// TIA Portal project "TP1200" (V15)
// HMI za 12' zaslon

(* hardware
DEVICE "HMI_1"  TP1200 Comfort
   slot 0: "HMI_1"  TP1200 Comfort  6AV2 124-0MC01-0AX0  15.0.0.0
   slot 1: "HMI_RT_1"  TP1200 Comfort  6AV2 124-0MC01-0AX0  15.0.0.0
   slot 5: "HMI_1.IE_CP_1"  PROFINET Interface  15.0.0.0
      slot 1: "PROFINET Interface_1"  PROFINET Interface
         slot 1: "Port_1"  Port
         slot 2: "Port_2"  Port
   slot 7: "HMI_1.MPI/DP_CP_1"  MPI/DP Interface  15.0.0.0
*)

(* ===== HMI "HMI_RT_1" =====
system functions are stored by id; their names below are inferred from use

HMI tags "Default tag table"
   "Tag_ScreenNumber" : UInt, internal

graphic list "PAH": 0 'PAHmiruje_2'; 1 'PAHdeluje_2'

graphic list "MOTOR_SMER": 0 'MotorNaprej_1'; 1 'MotorNazaj_1'

graphic list "MOTOR_ON_OFF": 0 'MotorON_1'; 1 'MotorOFF'

graphic list "NACINI_DELOVANJA": 0..1 'Nastavitev_2'; 2..3 'ROC_1'; 4..5 'ROC_CIKEL_1'; 6..7 'AVT_NOZNO_2'; 8..9 'AVT_2'

screen "Root screen" 1280x800, template "Template_2"
   on GenerateScreen: SetTag("Tag_ScreenNumber", 1)

Template "Template_2" 1280x800
   GraphicView "Template_Graphic view_1" at 0,0 size 1277x800; Picture "root_template_3"
   IOField "Template_I/O field_1" at 1111,2 size 165x94; FormatPattern 999
   TextField "Template_Text field_1" at 529,48 size 224x52; Text 'RPM'
   TextField "Template_Text field_2" at 988,4 size 85x52; Text 'Text'
   GraphicView "Template_Graphic view_3" at 19,118 size 436x567; Picture "bruderer logo_2"
   Button "Template_Button_11" at 637,689 size 131x109; TextOff 'Text'
      on Click: function_efd93a16("ANAL.VHODI", 477, 157, -1, -1, 2)
   IOField "Template_I/O field_2" at 554,2 size 164x92; FormatPattern 999
   IOField "Template_I/O field_3" at 717,2 size 402x93; FormatPattern 999999
   Button "Template_Button_12" at 893,689 size 131x109; TextOff 'Text'
      on Click: function_efd93a16("DEBELINA", 477, 157, -1, -1, 2)
   Button "Template_Button_13" at 507,688 size 131x109; TextOff 'Text'
      on Click: function_efd93a16("DIG.VHODi", 477, 157, -1, -1, 2)
   Button "Template_Button_14" at 765,688 size 131x109; TextOff 'Text'
      on Click: function_efd93a16("DIG.IZHODI", 477, 157, -1, -1, 2)
   Button "Template_Button_15" at 380,689 size 131x109; TextOff 'Text'
      on Click: function_efd93a16("HOD", 477, 157, -1, -1, 2)
   Button "Template_Button_16" at 254,690 size 131x109; TextOff 'Text'
      on Click: function_efd93a16("PODAJALNA", 477, 157, -1, -1, 2)
   Button "Template_Button_17" at 129,690 size 131x109; TextOff 'Text'
      on Click: function_efd93a16("PAH", 477, 157, -1, -1, 2)
   Button "Template_Button_18" at 1022,688 size 131x109; TextOff 'Text'
      on Click: function_efd93a16("PODATKI", 477, 157, -1, -1, 2)
   Button "Template_Button_19" at 1145,687 size 131x109; TextOff 'Text'
      on Click: function_efd93a16("LISTANAPAK", 477, 157, -1, -1, 2)
   TextField "Template_Text field_3" at 719,5 size 401x44; Text 'ŠIFRA IZDELKA'
   TextField "Template_Text field_4" at 1121,58 size 151x44; Text 'RPM'
   Button "Template_Button_1" at 0,690 size 131x109; TextOff 'Text'
      on Click: function_efd93a16("stevci", 477, 157, -1, -1, 2)
   GraphicIOField "Template_Graphic I/O field_2" at 0,0 size 311x94; PictureList "NACINI_DELOVANJA"
   IOField "Template_I/O field_5" at 304,2 size 257x50; FormatPattern ????
   IOField "Template_I/O field_4" at 304,49 size 258x44; FormatPattern 99999999999999999999999999999999
   GraphicIOField "Graphic I/O field_2" at 1144,155 size 135x134; PictureList "MOTOR_SMER"
   GraphicIOField "Graphic I/O field_1" at 1144,290 size 135x134; PictureList "MOTOR_SMER"
   GraphicIOField "Graphic I/O field_3" at 1144,425 size 135x134; PictureList "PAH"

PopupScreen "PODATKI" 650x510
   GraphicView "Graphic view_1" at 0,0 size 649x510; Picture "ParametriOrodja"
   TextField "Text field_1" at 17,169 size 152x47; Text 'OZNAKA'
   TextField "Text field_2" at 16,240 size 153x41; Text 'POMIK'
   TextField "Text field_3" at 15,307 size 153x44; Text 'HOD'
   TextField "Text field_4" at 15,371 size 155x49; Text 'VIŠINA ORODJA'
   TextField "Text field_5" at 389,375 size 152x43; Text 'HIT. PODAJANJA'
   TextField "Text field_6" at 390,302 size 156x49; Text 'POSPEŠEK'
   TextField "Text field_9" at 388,237 size 159x45; Text 'PODLOGA ZGORAJ'
   TextField "Text field_10" at 389,169 size 154x44; Text 'PODLOGA SPODAJ'
   TextField "Text field_11" at 17,439 size 155x49; Text 'SPROSITEV'

PopupScreen "PODAJALNA" 650x510
   GraphicView "Graphic view_1" at 0,0 size 649x510; Picture "PodajalnikTraku_1"

PopupScreen "PAH" 650x510
   GraphicView "Graphic view_1" at 0,0 size 649x510; Picture "VisinaPaha"

PopupScreen "LISTANAPAK" 650x510
   GraphicView "Graphic view_1" at 0,0 size 649x510; Picture "ListaNapak_2"

PopupScreen "HOD" 650x510
   GraphicView "Graphic view_1" at 0,0 size 649x510; Picture "HOD"

PopupScreen "DIG.VHODi" 650x510
   GraphicView "Graphic view_1" at 0,0 size 649x510; Picture "DI_1"

PopupScreen "DEBELINA" 650x510
   GraphicView "Graphic view_1" at 0,0 size 650x510; Picture "DI_KLASIKA_1"
   TextField "Text field_1" at 34,81 size 148x30; Text 'POMIK 1'
   TextField "Text field_2" at 40,311 size 151x30; Text 'POMIK 2'

PopupScreen "ANAL.VHODI" 650x510
   GraphicView "Graphic view_1" at 0,0 size 650x510; Picture "AI"

PopupScreen "DIG.IZHODI" 650x510
   GraphicView "Graphic view_1" at 1,0 size 649x510; Picture "DO_1"
   TextField "Text field_1" at 35,368 size 158x32; Text 'MAZANJE'
   TextField "Text field_2" at 34,300 size 157x35; Text 'IZPIHOVANJE'
   TextField "Text field_3" at 37,234 size 160x29; Text 'CAM2'
   TextField "Text field_4" at 33,163 size 161x38; Text 'CAM1'
   TextField "Text field_5" at 243,126 size 91x44; Text 'START'
   TextField "Text field_8" at 386,128 size 90x37; Text 'STOP'
   TextField "Text field_9" at 531,124 size 75x44; Text 'KORAK'

PopupScreen "stevci" 650x510
   TextField "Text field_5" at 213,64 size 210x50; Text 'NASTAVLJENO'
   TextField "Text field_1" at 6,125 size 200x61; Text 'ŠTEVEC SERIJE'
   TextField "Text field_2" at 6,196 size 200x61; Text 'SKUPAJ KOSOV 1'
   TextField "Text field_3" at 6,268 size 200x61; Text 'SKUPAJ KOSOV 2'
   TextField "Text field_4" at 6,346 size 200x64; Text 'KONEC SERIJE'
   TextField "Text field_15" at 434,64 size 210x50; Text 'IZDELANO'
   IOField "I/O field_1" at 211,124 size 210x64; FormatPattern 99999999999999999999999999
   IOField "I/O field_2" at 211,195 size 210x64; FormatPattern 99999999999999999999999999
   IOField "I/O field_3" at 211,268 size 210x64; FormatPattern 99999999999999999999999999
   IOField "I/O field_4" at 209,346 size 60x64; FormatPattern 9999
   IOField "I/O field_5" at 294,346 size 54x64; FormatPattern 99
   TextField "Text field_6" at 267,358 size 32x43; Text 'H'
   TextField "Text field_7" at 346,357 size 58x42; Text 'min'
   IOField "I/O field_6" at 434,124 size 210x64; FormatPattern 99999999999999999999999999
   IOField "I/O field_7" at 434,195 size 210x64; FormatPattern 99999999999999999999999999
   IOField "I/O field_8" at 434,268 size 210x64; FormatPattern 99999999999999999999999999
   TextField "Text field_8" at 401,349 size 131x61; Text 'FAKTOR'
   IOField "I/O field_9" at 537,347 size 107x64; FormatPattern 99
   Group "Group" at 6,64 size 638x347

PopupScreen "DEBELINA_KLASIKA" 650x535
   GraphicView "Graphic view_1" at 0,0 size 650x535; Picture "DI_KLASIKA_3"
*)